{attribute 'qualified_only'}
{attribute 'strict'}
TYPE E_SHUTTER_RPC_ERROR :
(
	OK					:= 0,
	NOT_OP				:= -1,			
	NOT_NOTOP_READY		:= -2,			
	NOT_NOTOP_NOTREADY	:= -3,			
	STILL_OPENING		:= -4,			
	STILL_CLOSING		:= -5,			
	LOCAL				:= -6			
);
END_TYPE

(* stored: Version 1.1.0.1, ProductVersion 3.1.4022.16
   DUT E_SHUTTER_RPC_ERROR: Id {ae0abd72-7773-43bc-83e5-11d973ea74e5} *)
